{attribute 'qualified_only'}
{attribute 'strict'}
TYPE SensorID :
(
	None := 1,
	Frontside := 2,
	Backside := 4
);
END_TYPE

(* stored: Version 1.1.0.1, ProductVersion 3.1.4024.12
   DUT SensorId: Id {1c42e517-6def-486c-82cc-002c428376f0} *)
